# EPICS StreamDevice protocol: protocols/s0ab.proto
Terminator = LF;
ExtraInput = Ignore;
ReplyTimeout = 4000;

setAbort {
        out "set_abort";
        in;
}
